Fanuc KAREL source: compact_preamble.KL

PROGRAM IO0209
%NOLOCKGROUP
ROUTINE RTEST
VAR
L1 : ARRAY[3] OF INTEGER;L2 : XYZWPR
L3 : JOINTPOS9
L4 : POSITION
A:BOOLEAN
S1:INTEGER
B:REAL
C:BOOLEAN
S2:REAL
BEGIN
A=TRUE
L1[1]=2
C=TRUE
S2=1.0
SET_REAL_REG(1,S2,S1)
END RTEST
BEGIN
RTEST
END IO0209
